// TIA Portal V17 export
// export: Created 2024-09-02T12:50:18.3547585Z, ExportSetting WithDefaults, DisplayName Totally Integrated Automation Portal, DisplayVersion V17, DisplayName TIA Portal Openness, DisplayVersion V17, DisplayName TIA Portal Version Control Interface, DisplayVersion V17, DisplayName STEP 7 Professional, DisplayVersion V17, DisplayName STEP 7 Safety, DisplayVersion V17, DisplayName WinCC Professional, DisplayVersion V17
DATA_BLOCK "LTLL_EKS_HMI_DATA_OP70"   // DB582
TITLE = LTLL_EksHmiData
{ S7_Optimized_Access := 'TRUE'; DB_Accessible_From_OPC_UA := 'FALSE' }
AUTHOR : Siemens
FAMILY : HMI_Lite
NAME : LTLL_EksHmiData
VERSION : 8.10
// stored: AutoNumber true, DBAccessibleFromOPCUA false, InstanceOfName LTLL_typeHmiEksData, InstanceOfType UDT, IsOnlyStoredInLoadMemory false, IsWriteProtectedInAS false
"LTLL_typeHmiEksData"
   // VAR
   //    eksAdapterIndex : UInt;
   //    costCenter : Array[0..3] of Char;
   //    dateEnd : Array[0..7] of Char;
   //    protectionLevel : Int;
   //    operatorID : Array[1..7] of Char;
   //    safetyMode : Byte;
   //    specialbits : Byte;
   //    serialNumber : Array[1..8] of Byte;
   //    keyAdapterReady : Bool;
   //    keyDetected : Bool;
   //    checksumNotOK : Bool;
   //    dateNotOK : Bool;
   //    costCenterNotOK : Bool;
   //    keyDataNotOK : Bool;
   //    eksKeyInvalidLess30Days : Bool;
   // END_VAR
BEGIN
END_DATA_BLOCK
